// TwinCAT 3 PLC project Stack
// ProgramVersion: 3.1.4026.11
// libraries:
//   Tc2_Standard, * (Beckhoff Automation GmbH)
//   Tc2_System, * (Beckhoff Automation GmbH)
//   [Resi4MPM], * (Jan Wilch)
//   [xPPU], * (Jan Wilch)
// project tree:
//   / HardwareContainer.TcPOU, MAIN.TcPOU, PlcTask.TcTTO
// (motion and I/O tree: see PLC project crane)
// real-time tasks:
//   TASK PlcTask: cycle T#10ms, priority 20, ADS port 350
//   TASK PlcTask1: cycle T#10ms, priority 23, ADS port 351
//   TASK PlcTask2: cycle T#10ms, priority 22, ADS port 352
//   TASK PlcTask3: cycle T#10ms, priority 21, ADS port 353
// variable links:
//   Stack/Stack Instance <-> Device (EtherCAT)/BK1 (EK1100)/1.10 (EL2004)
//     PlcTask Outputs/MAIN.m_panelMgr.DO_GreenLight <-> Channel 1/Output
//     PlcTask Outputs/MAIN.m_panelMgr.DO_WhiteLight <-> Channel 2/Output
//   Stack/Stack Instance <-> Device (EtherCAT)/BK1 (EK1100)/1.2 (EL1004)
//     PlcTask Inputs/MAIN.m_panelMgr.DI_EStopBtn <-> Channel 1/Input
//     PlcTask Inputs/MAIN.m_panelMgr.DI_ModeSwitch <-> Channel 3/Input
//     PlcTask Inputs/MAIN.m_panelMgr.DI_StartBtn <-> Channel 2/Input
//   Stack/Stack Instance <-> Device (EtherCAT)/BK1 (EK1100)/1.3 (EL1004)
//     PlcTask Inputs/MAIN.m_container.m_stack.o_slidingCylinder.DI_Extended <-> Channel 4/Input
//     PlcTask Inputs/MAIN.m_container.m_stack.o_slidingCylinder.DI_Retracted <-> Channel 3/Input
//   Stack/Stack Instance <-> Device (EtherCAT)/BK1 (EK1100)/1.4 (EL1004)
//     PlcTask Inputs/MAIN.m_container.m_stack.m_Inductivesensor.DI_WPMetallic <-> Channel 1/Input
//     PlcTask Inputs/MAIN.m_container.m_stack.m_Opticalsensor.DI_WPLight <-> Channel 2/Input
//   Stack/Stack Instance <-> Device (EtherCAT)/BK1 (EK1100)/1.5 (EL1004)
//     PlcTask Inputs/MAIN.m_container.m_stack.m_Presencesensor.DI_WPDetected <-> Channel 2/Input
//   Stack/Stack Instance <-> Device (EtherCAT)/BK1 (EK1100)/1.9 (EL2004)
//     PlcTask Outputs/MAIN.m_container.m_stack.o_slidingCylinder.DO_Extend <-> Channel 2/Output
//   Stack/Stack Instance <-> Device (EtherCAT)/BK4 (EK1100)/4.3 (EL1004)
//     PlcTask Inputs/MAIN.m_container.m_stack.o_slidingCylinder.DI_BoundaryPressure <-> Channel 1/Input
//   Stack/Stack Instance <-> Device (EtherCAT)/BK6 (EK1100)/6.2 (EL3062)
//     PlcTask Inputs/MAIN.m_container.m_stack.m_Weightsensor.AI_WPWeight <-> AI Standard Channel 1/Value

CONFIGURATION Stack
    RESOURCE PLC ON TwinCAT3
        TASK PlcTask(INTERVAL := T#10ms, PRIORITY := 22);
        PROGRAM MAIN WITH PlcTask : MAIN;
    END_RESOURCE
END_CONFIGURATION

// ---- MAIN.TcPOU
PROGRAM MAIN
VAR CONSTANT
	IGNORE_DEFINITION: BOOL := TRUE;
END_VAR
VAR
	m_errorManager: ErrorManager;
	m_services: ServiceContainer(ADR(m_errorManager));
	
	m_panelMgr: PanelManager(
		m_services.PtrStateTracker,
		EProcessVariables.Pnl_Stack_Start,
		0,
		EProcessVariables.Pnl_Stack_Mode,
		EProcessVariables.Pnl_Stack_EStop,
		0);
	
	// instantiate machine behavior model
	m_container: HardwareContainer(
		m_services.PtrStateTracker, 
		m_services.PtrProcessManager, 
		ADR(m_errorManager));
	
	m_modes: MachineModes(ADR(m_services), ADR(m_panelMgr));
	
	m_appObservation: ARRAY[EProcessVariables.OpMode_Stack..EProcessVariables.OpMode_Stack] OF SValue;

	// TESTING
// 	m_lscConnected: BOOL;
// 	m_craneConnected: BOOL;
// 	m_stackConnected: BOOL;
// 	m_stampConnected: BOOL;
END_VAR

// process state observation
m_appObservation[EProcessVariables.OpMode_Stack].DataType := EDataType.string_t;
m_appObservation[EProcessVariables.OpMode_Stack].Value.String_t := m_modes.SFCCurrentStep;
m_appObservation[EProcessVariables.OpMode_Stack].Defined := TRUE;

// cylic service updates
m_services.PtrStateTracker^.CyclicUpdateStatus(IGNORE_DEFINITION, m_appObservation);
m_services.PtrProcessManager^.CyclicManageBehavior();

// main state machine
m_modes();

// TESTING
// IF m_services.PtrStateTracker^.GetString(EProcessVariables.OpMode_LSC) <> '' THEN
// 	m_lscConnected := TRUE;
// END_IF
// IF m_services.PtrStateTracker^.GetString(EProcessVariables.OpMode_Stack) <> '' THEN
// 	m_stackConnected := TRUE;
// END_IF
// IF m_services.PtrStateTracker^.GetString(EProcessVariables.OpMode_Stamp) <> '' THEN
// 	m_stampConnected := TRUE;
// END_IF
// IF m_services.PtrStateTracker^.GetString(EProcessVariables.OpMode_Crane) <> '' THEN
// 	m_craneConnected := TRUE;
// END_IF

END_PROGRAM

// ---- HardwareContainer.TcPOU
FUNCTION_BLOCK HardwareContainer
VAR
	// hardware control POUs
	m_stack: Stack;
	m_indic: ActivityIndicator(i_signalProcVar := EProcessVariables.Test_StackFree);
	
	// products
	{attribute 'OPC.UA.DA' := '1'}
	{attribute 'OPC.UA.DA.Access' := '1'}
	m_stackWP: xPPUProduct(EProcessVariables.Stack_ProductType, EProcessVariables.Stack_ProductStamped);
	
	// hardware observation (if not included in hardware control)
	m_observeStack: ObserveStack(ADR(m_stack), ADR(m_stackWP));
	
	// control primitives
	m_stackProvide: Stack_ProvideWorkpiece(ADR(m_stack));
	m_delay: Delay;
	m_indicCP_Stack: IndicateActivity(i_id := EPrimitives.Gen_IndicateActive_Stack, i_ptrIndicator := ADR(m_indic));
	m_forceVal_Stack: ForceProcessVariable(i_id := EPrimitives.Gen_ForceVariable_Stack);
	
	// module sequences
END_VAR

METHOD FB_init : BOOL
VAR_INPUT
	bInitRetains : BOOL; // if TRUE, the retain variables are initialized (warm start / cold start)
	bInCopyCode : BOOL;  // if TRUE, the instance afterwards gets moved into the copy code (online change)

	i_ptrStateTracker: POINTER TO StateTracker;
	i_ptrProcessManager: POINTER TO ProcessManager;
	
	i_ptrErrorManager: POINTER TO ErrorManagerBase;
END_VAR
m_stackProvide.ProvideServices(i_ptrProcessManager, i_ptrStateTracker);
m_delay.ProvideServices(i_ptrProcessManager, i_ptrStateTracker);
m_indicCP_Stack.ProvideServices(i_ptrProcessManager, i_ptrStateTracker);
m_forceVal_Stack.ProvideServices(i_ptrProcessManager, i_ptrStateTracker);

// provide Behaviors to the Process Manager
i_ptrProcessManager^.AddPrimitive(ADR(m_stackProvide));
i_ptrProcessManager^.AddPrimitive(ADR(m_delay));
i_ptrProcessManager^.AddPrimitive(ADR(m_indicCP_Stack));
i_ptrProcessManager^.AddPrimitive(ADR(m_forceVal_Stack));

// provide observations to the Process Manager
i_ptrStateTracker^.AddObservation(ADR(m_observeStack));
i_ptrStateTracker^.AddObservation(ADR(m_indic));

// provide workpieces to the Process Manager
i_ptrStateTracker^.RegisterLocalProduct(EProducts.stack_product, ADR(m_stackWP));
END_METHOD

END_FUNCTION_BLOCK
